FUNCTION_BLOCK FB_Home_Z
(*========================================
Execute需一直有效，功能块才会一直执行
先回原点，然后直接到等待位
==========================================*)
VAR_IN_OUT
	Axis				:AXIS_REF;	(* B *)
END_VAR
VAR_INPUT
	Execute				:BOOL;	(* B *)
	PosLimit			:BOOL;			(*正极限位信号*)
	NegLimit			:BOOL;			(*负极限位信号*)
	Position			:LREAL			(* B *) := DEFAULT_HOME_POSITION;
	HomeingVelo			:LREAL:=5;
	Standby_position	:LREAL;		//最终待机位
	bCalibrationCam 	:BOOL;	(* V *)	(* Beckhoff proprietary input *)
	rel_dis         	:LREAL:=10;  //碰到原点后，正向移动距离，在开始寻原点
	TimeOutSet       	:LREAL;//s
	reset				:BOOL;
	maxDistance:LREAL;
END_VAR
VAR_OUTPUT
	Done				:BOOL;	(* B *)
	Busy				:BOOL;	(* E *)
	Active				:BOOL;	(* E *)
	CommandAborted		:BOOL;	(* E *)
	Error				:BOOL;	(* B *)
	ErrorID				:UDINT;	(* E *)
	TimeOut				:BOOL;//回零超时
	HomeErr				:BOOL;//超过最大行程

END_VAR
VAR
	mcJog			:MC_Jog;
	mcHome			:MC_Home;
	mcRel           :MC_MoveRelative;
	mcAbs           :MC_MoveAbsolute;	
	mcStop			:MC_Stop;
	HomeStep		:INT;
	ton				:TON;
	StopDo			:BOOL;
	start_pos		:LREAL;
	start_r_trig:Tc2_Standard.R_TRIG;
END_VAR

ton(IN:=Execute , PT:=LREAL_TO_TIME(TimeOutSet*1000) , Q=> , ET=> );
IF ton.Q THEN 
	TimeOut:=TRUE;
	HomeStep	:=100;
END_IF

start_r_trig(CLK:=Execute , Q=> );
IF start_r_trig.Q THEN 
	start_pos:=Axis.NcToPlc.ActPos;
END_IF


IF  NOT Execute THEN
	mcJog.JogForward		:=FALSE;
	mcJog.JogBackwards		:=FALSE;
	mcHome.Execute			:=FALSE;
	mcRel.Execute			:=FALSE;
	mcAbs.Execute			:=FALSE;
	done					:=FALSE;
	busy					:=FALSE;	
	HomeStep				:=0;
END_IF

IF reset THEN 
	Error					:=FALSE;
	TimeOut					:=FALSE;
	HomeErr			:=FALSE;
END_IF

CASE HomeStep OF

0:
	busy	:=FALSE;
	Done	:=FALSE;
	IF 	Execute AND NOT Error  THEN		
		IF  NOT bCalibrationCam THEN
			HomeStep	:=10;
		ELSE
			HomeStep	:=20;
		END_IF
		busy	:=TRUE;
		ErrorID	:=0;		
	END_IF
	
10:(*先向负限位方向运动*)
	mcJog.JogForward		:=FALSE;
	mcJog.JogBackwards		:=TRUE;		 
	IF	bCalibrationCam THEN
		mcJog.JogBackwards	:=FALSE;		
		HomeStep	:=20;		
	ELSIF mcJog.Error   THEN
			HomeStep	:=100;
	ELSIF ABS(start_pos-Axis.NcToPlc.ActPos)>maxDistance THEN 
			HomeStep	:=100;
			HomeErr:=TRUE;
	END_IF
	
20:(*从原点处正方向移动一段距离*)
	mcRel.Execute		:=TRUE;	
	IF mcRel.Done AND Axis.Status.NotMoving THEN 
		mcRel.Execute	:=FALSE;
		HomeStep		:=30;
	ELSIF mcRel.Error OR TimeOut THEN 
		HomeStep	:=100;	
	END_IF
	
30:(*调用回零功能块*)
	mcHome.Execute	:=TRUE;
	IF mcHome.Done AND AXIS.Status.Homed THEN
		mcHome.Execute	:=FALSE;		
		HomeStep		:=50;
	ELSIF AXIS.Status.Error OR TimeOut THEN
		HomeStep		:=100;
	END_IF
(*	
40:(*碰正极限*)
	mcJog.JogBackwards		:=FALSE;
	mcJog.JogForward		:=TRUE;		(*向正限位方向运动*)	
	IF PosLimit THEN 
		mcJog.JogForward	:=FALSE;
		IF Axis.Status.NotMoving THEN
			HomeStep	:=50;
		END_IF
	ELSIF mcJog.Error OR TimeOut THEN
			HomeStep	:=100; 
	END_IF
*)	
50:(*回待机位*)
	mcAbs.Execute:=TRUE;
	IF mcAbs.Done AND Axis.Status.NotMoving THEN 
		mcAbs.Execute	:=FALSE;
		done			:=TRUE;
		HomeStep		:=99; 		
	END_IF
99:
	;	

100:
	Error			:=TRUE;
	IF	mcHome.ErrorID <> 0 THEN
		ErrorID			:=mcHome.ErrorID;
	ELSIF  mcJog.ErrorID <> 0 THEN
		ErrorID			:=mcJog.ErrorID;
	ELSIF mcRel.ErrorID<>0 THEN 
		ErrorID			:=mcRel.ErrorID;
	ELSIF mcAbs.ErrorID<>0 THEN 
		ErrorID			:=mcAbs.ErrorID;	
	END_IF
	mcJog.JogForward		:=FALSE;
	mcJog.JogBackwards		:=FALSE;
	mcHome.Execute			:=FALSE;
	mcRel.Execute			:=FALSE;
	mcAbs.Execute			:=FALSE;
	StopDo			:=TRUE;
	HomeStep		:=0;
	
END_CASE


Call_FB();

ACTION Call_FB:
Axis.ReadStatus();
mcJog
	(
	Velocity:=	HomeingVelo ,
	Mode:=		MC_JOGMODE_CONTINOUS ,
	Axis:=		Axis ,
	);

mcHome
	(
	Execute:= ,
	Position:=			Position ,
	HomingMode:= 		,
	BufferMode:= 		,
	Options:=			 ,
	bCalibrationCam:=	bCalibrationCam ,
	Axis:=				Axis ,
	);

mcRel(
	Axis:=Axis , 
	Execute:= , 
	Distance:=rel_dis , 
	Velocity:= HomeingVelo, 
	Acceleration:= , 
	Deceleration:= , 
	Jerk:= , 
	BufferMode:= , 
	Options:= , 
	Done=> , 
	Busy=> , 
	Active=> , 
	CommandAborted=> , 
	Error=> , 
	ErrorID=> );
mcAbs(
	Axis:=Axis , 
	Execute:= , 
	Position:=Standby_position , 
	Velocity:=HomeingVelo , 
	Acceleration:= , 
	Deceleration:= , 
	Jerk:= , 
	BufferMode:= , 
	Options:= , 
	Done=> , 
	Busy=> , 
	Active=> , 
	CommandAborted=> , 
	Error=> , 
	ErrorID=> );
mcStop(
	Axis:=Axis , 
	Execute:=StopDo , 
	Deceleration:= , 
	Jerk:= , 
	Options:= , 
	Done=> , 
	Busy=> , 
	Active=> , 
	CommandAborted=> , 
	Error=> , 
	ErrorID=> );
IF mcStop.Busy THEN 
	StopDo:=FALSE;
END_IF
END_ACTION

END_FUNCTION_BLOCK

(* stored: Version 1.1.0.1, ProductVersion 3.1.4024.11
   POU FB_Home_Z: Id {bb160ba1-c2c3-4fad-9357-e04ea5be8426}, SpecialFunc None
   Action Call_FB: Id {d40449a3-0e85-4a44-9180-9ba27d63e5ce} *)
